{attribute 'Tc2GvlVarNames'}
VAR_CONFIG
END_VAR

(* stored: Version 1.1.0.1, ProductVersion 3.1.4020.6
   GVL Variablen_Konfiguration: Id {3af5dee9-c3e8-442f-9917-da7acdaeecbb} *)
